// Mitsubishi GX Works2 project: PLC_GROUP9   PLC: FX3G

// global labels: Global1
VAR_GLOBAL
  init AT X010 : BOOL;
END_VAR
VAR_GLOBAL CONSTANT
  OrangeValue : REAL;
END_VAR
VAR_GLOBAL
  RE_initOrange AT D1100 : REAL;
END_VAR
VAR_GLOBAL CONSTANT
  ClementineValue : REAL;
END_VAR
VAR_GLOBAL
  RE_initClem AT D1120 : REAL;
END_VAR
VAR_GLOBAL CONSTANT
  PomeloValue : REAL;
END_VAR
VAR_GLOBAL
  RE_initPomeo AT D1110 : REAL;
  Sw10 AT X010 : BOOL;
END_VAR
VAR_GLOBAL CONSTANT
  CorrectDiv : INT := 2;
END_VAR
VAR_GLOBAL
  RE_CorrectDiv AT D1115 : REAL;
END_VAR
VAR_GLOBAL CONSTANT
  HelpValue : INT := 1;
END_VAR
VAR_GLOBAL
  StopWork AT X007 : BOOL;
END_VAR
VAR_GLOBAL CONSTANT
  two : REAL := 2.0;
END_VAR
VAR_GLOBAL
  ClementineOn AT M0 : BOOL;
  PomeloOn AT M1 : BOOL;
  bulb1 AT Y010 : BOOL;
END_VAR
VAR_GLOBAL CONSTANT
  zero : REAL;
END_VAR
VAR_GLOBAL
  RE_Orange AT D1150 : REAL;
  RE_Clem AT D1130 : REAL;
  RE_Pomelo AT D1140 : REAL;
  SystemOn AT M2 : BOOL;
  bnnb AT M3 : BOOL;
  m_6 AT M7 : BOOL;
  StartingValuesOn AT M0 : BOOL;
  InventoryValuesOn AT M1 : BOOL;
  SystemOff AT M2 : BOOL;
  SystemOf AT M2 : BOOL;
  StopConditions AT M3 : BOOL;
  FlashingLight1 AT M4 : BOOL;
  FlickeringTimer1 AT TC0 : BOOL;
END_VAR
VAR_GLOBAL CONSTANT
  VNBVNBV : INT := 30;
  ConstantFlickering1 : INT := 5;
END_VAR
VAR_GLOBAL
  TimerValue1 AT TS0 : BOOL;
  FlickeringLight1 AT M4 : BOOL;
  FlickeringLight2 AT M5 : BOOL;
  FlickeringTimer2 AT TC1 : BOOL;
  TimerValue2 AT TS1 : BOOL;
  FlickeringLightStop AT M6 : BOOL;
  FlickeringTimer3 AT TC2 : BOOL;
  FlickeringStoper AT TS2 : BOOL;
END_VAR
VAR_GLOBAL CONSTANT
  Var_Time_0 : INT := 30;
END_VAR
VAR_GLOBAL
  Constant_300 AT K3 : INT;
  Washing_help AT M10 : BOOL;
  Start AT M10 : BOOL;
  Start_Washing AT X002 : BOOL;
  light_on AT M11 : BOOL;
  Close_light AT TS3 : BOOL;
  Start_light AT M10 : BOOL;
  bulb5 AT Y005 : BOOL;
  Start_Wash AT M10 : BOOL;
END_VAR
VAR_GLOBAL CONSTANT
  Constant_100 : REAL := 100;
END_VAR
VAR_GLOBAL
  More_100 AT M12 : BOOL;
  Washing_Orange AT D1170 : REAL;
  over_100_ans AT M13 : BOOL;
END_VAR
VAR_GLOBAL CONSTANT
  Constant_2 : REAL := 2;
END_VAR
VAR_GLOBAL
  Quantity_To_Move AT D1180 : REAL;
  Finish_Orange AT M15 : BOOL;
  Washing_Clem AT D1190 : REAL;
  Washing_Pomalo AT D1200 : REAL;
  under_100_ans AT M14 : BOOL;
  orange_ans AT M13 : BOOL;
END_VAR
VAR_GLOBAL CONSTANT
  ConstantFlickering : INT := 30;
END_VAR
VAR_GLOBAL
  StartCounter AT CC0 : BOOL;
END_VAR
VAR_GLOBAL CONSTANT
  CounterStert : INT := 3;
  CounterStart : INT := 1;
END_VAR
VAR_GLOBAL
  StertDay AT CS0 : BOOL;
  not1 AT M30 : BOOL;
  not2 AT M31 : BOOL;
  Timer3 AT TC3 : BOOL;
END_VAR
VAR_GLOBAL CONSTANT
  ConstantWashing : INT := 30;
END_VAR
VAR_GLOBAL
  End_level1 AT M16 : BOOL;
END_VAR
VAR_GLOBAL CONSTANT
  DubbleClick : INT := 2;
END_VAR
VAR_GLOBAL
  Start_level_Two AT CC1 : BOOL;
  Start_Collect AT X001 : BOOL;
  Start_Collect_SW AT X011 : BOOL;
  Collect_light AT Y001 : BOOL;
  Squeeze_SW AT X011 : BOOL;
  Squeezing : BOOL;
  Start_squeezing AT CS1 : BOOL;
  Start_level_Three AT CC1 : BOOL;
  SqueezeContainer AT D2200 : REAL;
  Finish_move AT M17 : BOOL;
  End_level2 AT M18 : BOOL;
  helpBulb AT M19 : BOOL;
  helpBulb2 AT M20 : BOOL;
  level_Three AT CS1 : BOOL;
  kkkk AT Y002 : BOOL;
  Timer4 AT TC4 : BOOL;
  Stop_Flickering AT TS4 : BOOL;
  SqueezeLight1 AT Y002 : BOOL;
  SqueezeLight2 AT Y003 : BOOL;
  JoiceContainer AT D1210 : REAL;
  JuiceContainer AT D1210 : REAL;
  End_level3 AT M32 : BOOL;
  helpBulb3 AT M41 : BOOL;
  Start_level_four AT X003 : BOOL;
  helpBulb4 AT M34 : BOOL;
  Start_Quality_Check AT X003 : BOOL;
  Failed_Check AT M38 : BOOL;
  Start_level_4 AT M35 : BOOL;
  Finish_level_three AT M40 : BOOL;
  Secend_Check AT CS5 : BOOL;
  Counter_Check AT CC5 : BOOL;
END_VAR
VAR_GLOBAL CONSTANT
  Limit_Check : INT := 2;
END_VAR
VAR_GLOBAL
  analog_input_2 AT D8281 : INT;
  analog_val AT D1300 : INT;
END_VAR
VAR_GLOBAL CONSTANT
  Constant_1 : INT := 1;
END_VAR
VAR_GLOBAL
  helpBulb6 AT M37 : BOOL;
END_VAR
VAR_GLOBAL CONSTANT
  Constant_5 : INT := 4;
END_VAR
VAR_GLOBAL
  helpBulbEnd3 AT M33 : BOOL;
  need_restart AT M39 : BOOL;
  FlickeringStoper5 AT TS5 : BOOL;
  Val_In_Range AT Y004 : BOOL;
  FlickeringTimer5 AT TC5 : BOOL;
END_VAR
VAR_GLOBAL CONSTANT
  ConstantFlickering5 : INT := 50;
END_VAR
VAR_GLOBAL
  Start_Container AT M41 : BOOL;
  Storage_Container AT D1320 : REAL;
  End_level4 AT M42 : BOOL;
  End_day AT M31 : BOOL;
  MoreThen1 AT M44 : BOOL;
  LessThen5 AT M45 : BOOL;
  ValBulb AT M46 : BOOL;
  Stoper AT CS0 : BOOL;
  endBulb1 AT M47 : BOOL;
  endBulb2 AT M48 : BOOL;
  endBulb3 AT M49 : BOOL;
  endBulb4 AT M50 : BOOL;
  Endbulb5 AT M51 : BOOL;
END_VAR
VAR_GLOBAL CONSTANT
  Constant_3c : REAL := 20;
END_VAR
VAR_GLOBAL
  Enough_Liter AT M57 : BOOL;
END_VAR
VAR_GLOBAL CONSTANT
  Constant_3 : REAL := 20;
END_VAR
VAR_GLOBAL
  Analog_Output AT D8282 : INT;
  Finish_Count AT M62 : BOOL;
  FlickeringTimer6 AT TC6 : BOOL;
  FlickeringStoper6 AT TS6 : BOOL;
  StartToBottle AT X006 : BOOL;
  End_level5 AT M60 : BOOL;
  notEnoughJuice AT M61 : BOOL;
  Timer6 AT TC6 : BOOL;
  StoperTimer6 AT TS6 : BOOL;
  NotBottle AT Y006 : BOOL;
END_VAR
VAR_GLOBAL CONSTANT
  ConvertingCon : INT := 404;
  Constant_10c : REAL := 20;
  Constant_20c : REAL := 20;
END_VAR
VAR_GLOBAL
  bulb1ForRest AT M70 : BOOL;
  bulb2ForRest AT M71 : BOOL;
  CheckStartCon AT M72 : BOOL;
  QuantityPerIteration AT D1340 : REAL;
  StartContainer AT CC0 : BOOL;
  StartToContainer AT X006 : BOOL;
  NotContainer AT Y006 : BOOL;
END_VAR
VAR_GLOBAL CONSTANT
  notEnough : INT;
END_VAR

// task Task_01 (event TRUE, interval 0, priority 31): POU_01

PROGRAM POU_01
(* structured ladder/FBD written out as ST: instructions are called as NAME(EN, inputs, outputs); _pN, _eN, _tN stand for wires *)
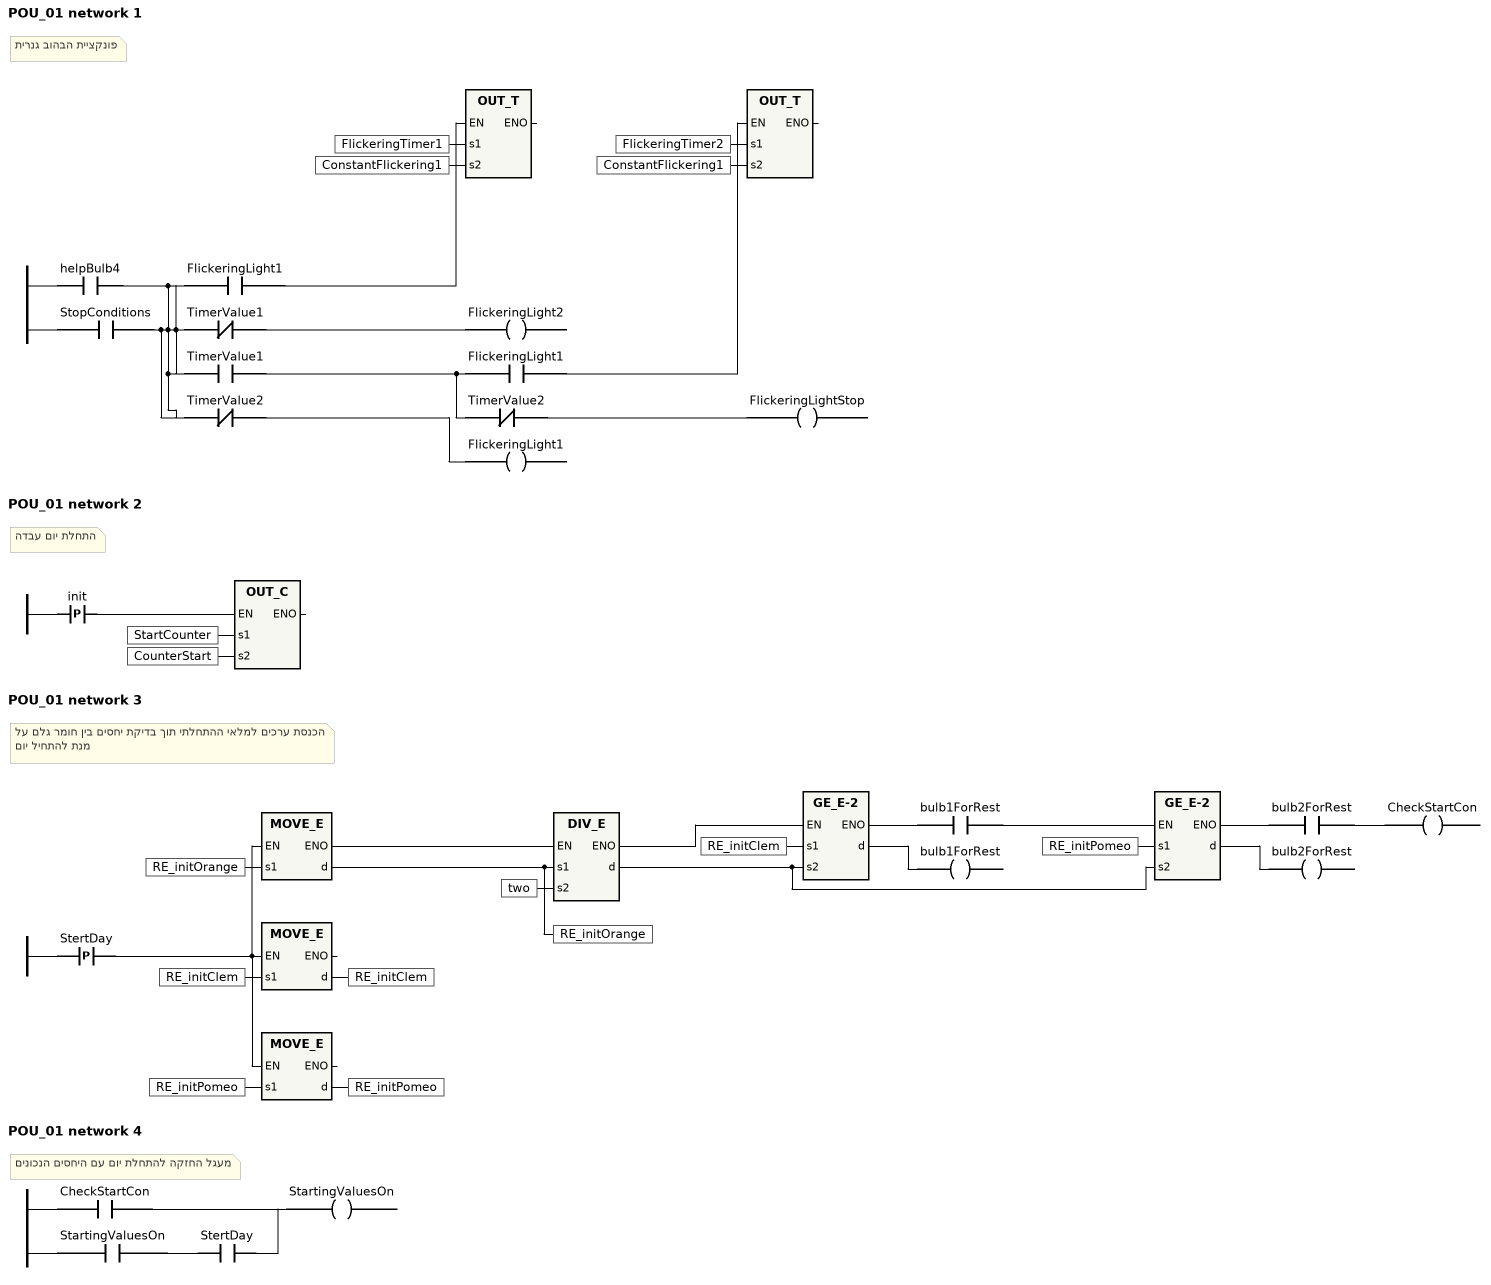
(* network 1 *)
(* פונקציית הבהוב גנרית *)
_p1 := helpBulb4 OR StopConditions;
OUT_T(_p1 AND FlickeringLight1, FlickeringTimer1, ConstantFlickering1);
FlickeringLight2 := _p1 AND NOT TimerValue1;
_p2 := _p1 AND TimerValue1;
OUT_T(_p2 AND FlickeringLight1, FlickeringTimer2, ConstantFlickering1);
FlickeringLightStop := _p2 AND NOT TimerValue2;
FlickeringLight1 := _p1 AND NOT TimerValue2;
(* network 2 *)
(* התחלת יום עבדה *)
OUT_C(LDP(TRUE, init), StartCounter, CounterStart);
(* network 3 *)
(* הכנסת ערכים למלאי ההתחלתי תוך בדיקת יחסים בין חומר גלם על מנת להתחיל יום *)
_p1 := LDP(TRUE, StertDay);
_e2 := MOVE_E(_p1, RE_initOrange, RE_initOrange);
_e4 := DIV_E(_e2, RE_initOrange, two, _t3);
_e6 := GE_E(_e4, RE_initClem, _t3, _t5);
bulb1ForRest := _t5;
MOVE_E(_p1, RE_initClem, RE_initClem);
_e8 := GE_E(_e6 AND bulb1ForRest, RE_initPomeo, _t3, _t7);
CheckStartCon := _e8 AND bulb2ForRest;
MOVE_E(_p1, RE_initPomeo, RE_initPomeo);
bulb2ForRest := _t7;
(* network 4 *)
(* מעגל החזקה להתחלת יום עם היחסים הנכונים *)
StartingValuesOn := CheckStartCon OR (StartingValuesOn AND StertDay);
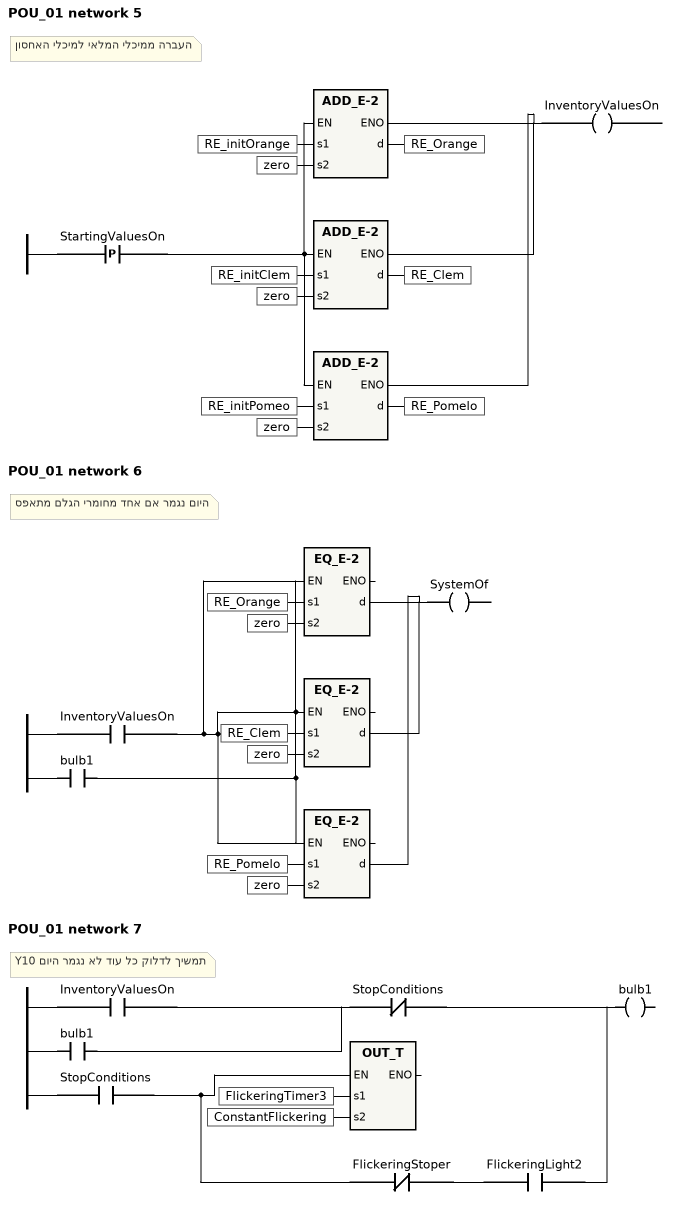
(* network 5 *)
(* העברה ממיכלי המלאי למיכלי האחסון *)
_p1 := LDP(TRUE, StartingValuesOn);
_e2 := ADD_E(_p1, RE_initOrange, zero, RE_Orange);
_e3 := ADD_E(_p1, RE_initClem, zero, RE_Clem);
_e4 := ADD_E(_p1, RE_initPomeo, zero, RE_Pomelo);
InventoryValuesOn := _e2 OR _e3 OR _e4;
(* network 6 *)
(* היום נגמר אם אחד מחומרי הגלם מתאפס *)
_p1 := InventoryValuesOn OR bulb1;
EQ_E(_p1, RE_Orange, zero, _t2);
EQ_E(_p1, RE_Clem, zero, _t3);
EQ_E(_p1, RE_Pomelo, zero, _t4);
SystemOf := _t2 OR _t3 OR _t4;
(* network 7 *)
(* תמשיך לדלוק כל עוד לא נגמר היום Y10 *)
bulb1 := ((InventoryValuesOn OR bulb1) AND NOT StopConditions) OR (StopConditions AND NOT FlickeringStoper AND FlickeringLight2);
OUT_T(StopConditions, FlickeringTimer3, ConstantFlickering);
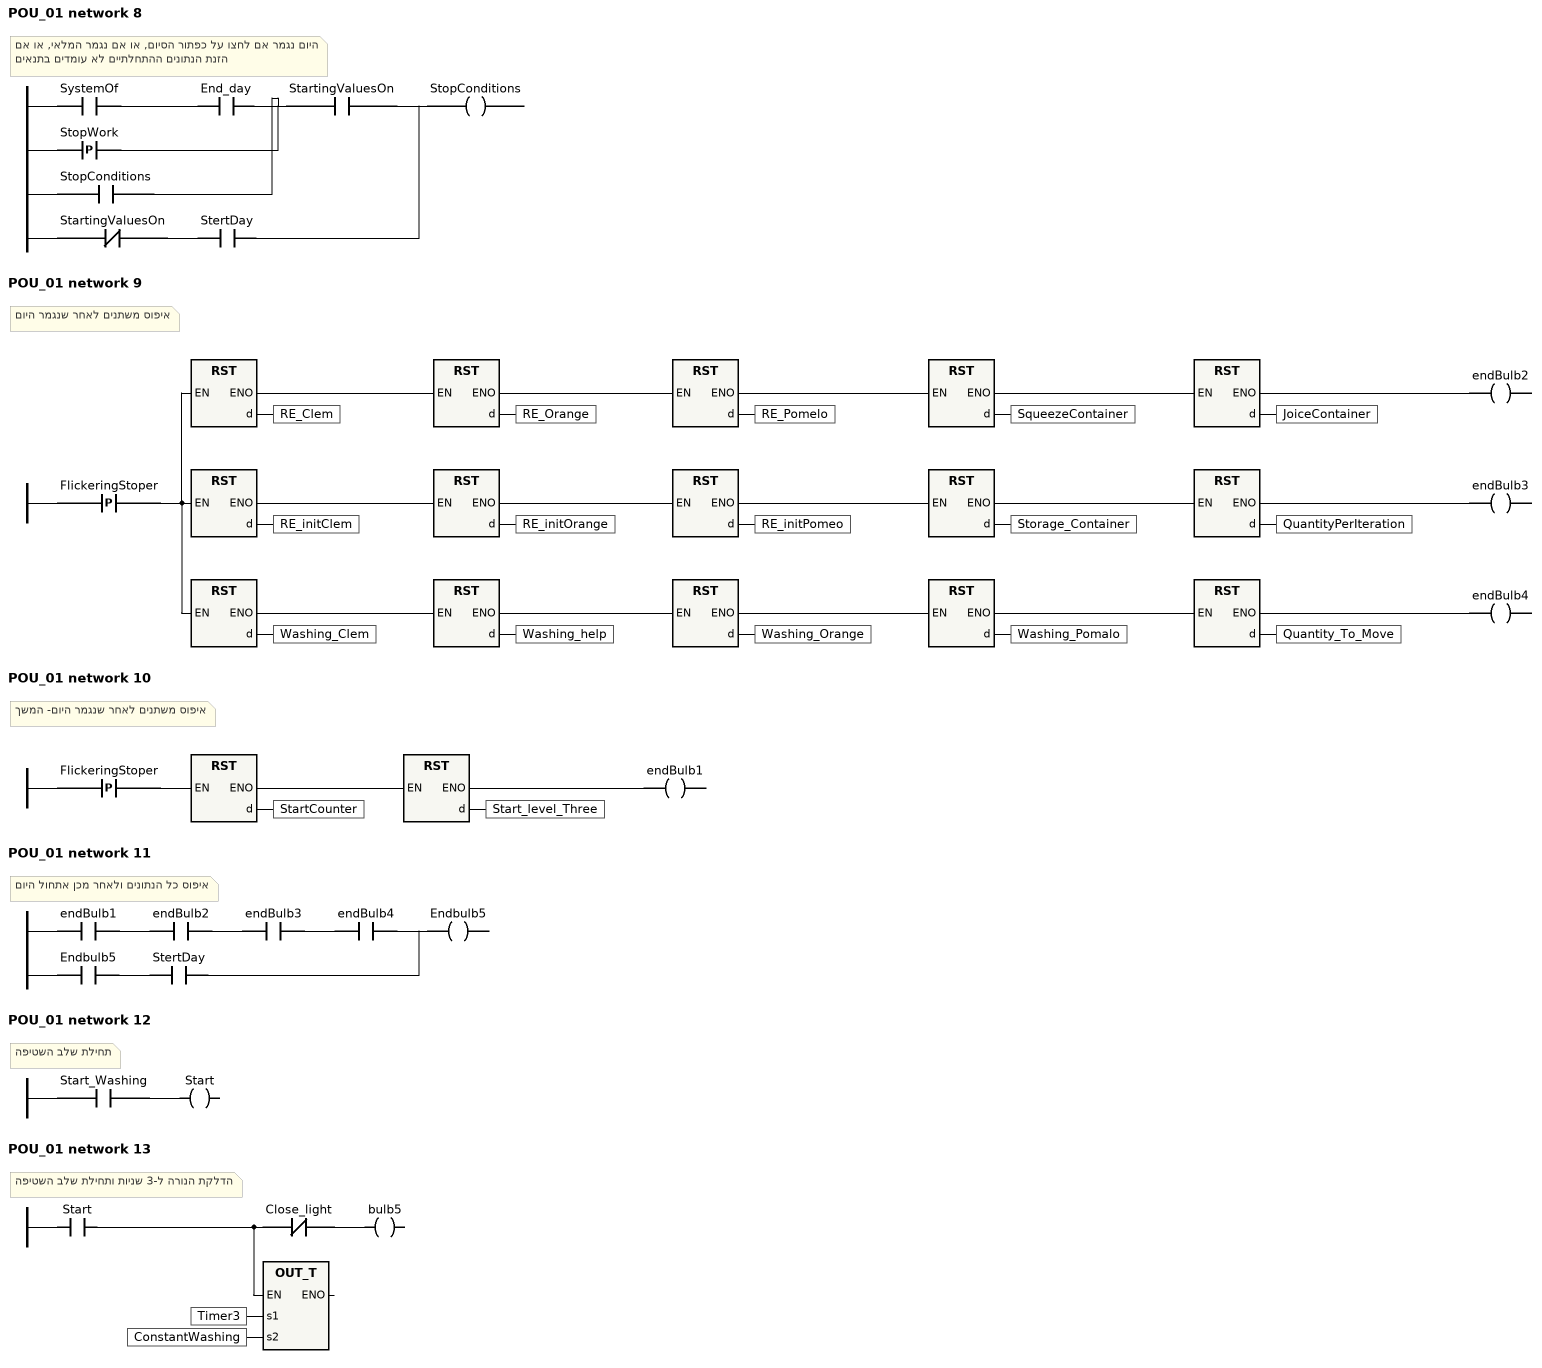
(* network 8 *)
(* היום נגמר אם לחצו על כפתור הסיום, או אם נגמר המלאי, או אם הזנת הנתונים ההתחלתיים לא עומדים בתנאים *)
StopConditions := (((SystemOf AND End_day) OR LDP(TRUE, StopWork) OR StopConditions) AND StartingValuesOn) OR (NOT StartingValuesOn AND StertDay);
(* network 9 *)
(* איפוס משתנים לאחר שנגמר היום *)
_p1 := LDP(TRUE, FlickeringStoper);
_e2 := RST(_p1, RE_Clem);
_e3 := RST(_e2, RE_Orange);
_e4 := RST(_e3, RE_Pomelo);
_e5 := RST(_e4, SqueezeContainer);
_e6 := RST(_e5, JoiceContainer);
endBulb2 := _e6;
_e7 := RST(_p1, RE_initClem);
_e8 := RST(_e7, RE_initOrange);
_e9 := RST(_e8, RE_initPomeo);
_e10 := RST(_e9, Storage_Container);
_e11 := RST(_e10, QuantityPerIteration);
endBulb3 := _e11;
_e12 := RST(_p1, Washing_Clem);
_e13 := RST(_e12, Washing_help);
_e14 := RST(_e13, Washing_Orange);
_e15 := RST(_e14, Washing_Pomalo);
_e16 := RST(_e15, Quantity_To_Move);
endBulb4 := _e16;
(* network 10 *)
(* איפוס משתנים לאחר שנגמר היום- המשך *)
_e1 := RST(LDP(TRUE, FlickeringStoper), StartCounter);
_e2 := RST(_e1, Start_level_Three);
endBulb1 := _e2;
(* network 11 *)
(* איפוס כל הנתונים ולאחר מכן אתחול היום *)
Endbulb5 := (endBulb1 AND endBulb2 AND endBulb3 AND endBulb4) OR (Endbulb5 AND StertDay);
(* network 12 *)
(* תחילת שלב השטיפה *)
Start := Start_Washing;
(* network 13 *)
(* הדלקת הנורה ל-3 שניות ותחילת שלב השטיפה *)
bulb5 := Start AND NOT Close_light;
OUT_T(Start, Timer3, ConstantWashing);
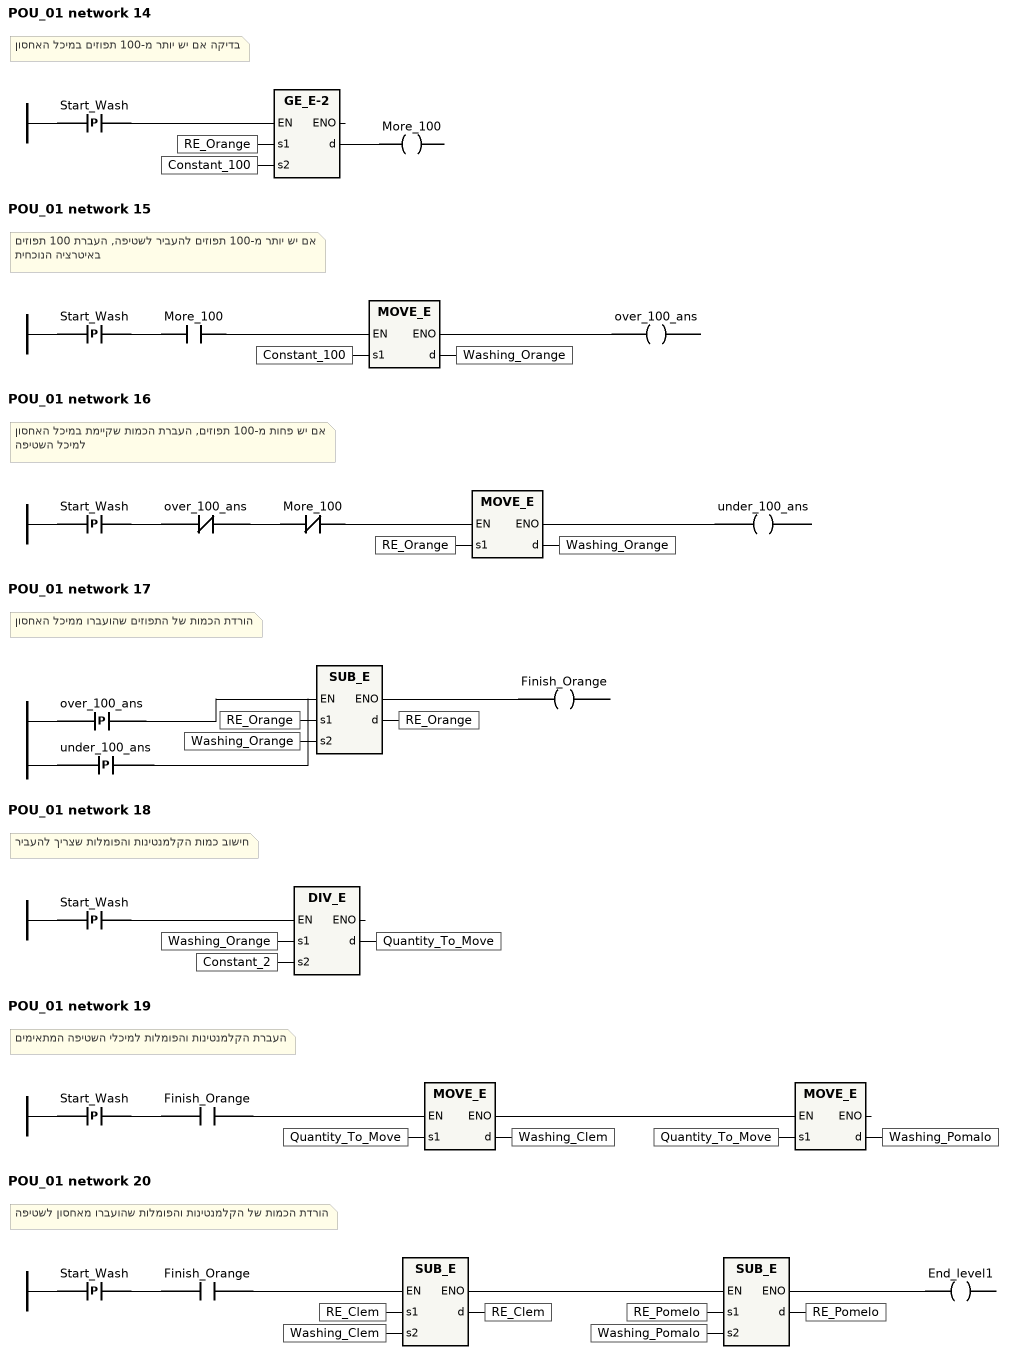
(* network 14 *)
(* בדיקה אם יש יותר מ-100 תפוזים במיכל האחסון *)
GE_E(LDP(TRUE, Start_Wash), RE_Orange, Constant_100, _t1);
More_100 := _t1;
(* network 15 *)
(* אם יש יותר מ-100 תפוזים להעביר לשטיפה, העברת 100 תפוזים באיטרציה הנוכחית *)
_e1 := MOVE_E(LDP(TRUE, Start_Wash) AND More_100, Constant_100, Washing_Orange);
over_100_ans := _e1;
(* network 16 *)
(* אם יש פחות מ-100 תפוזים, העברת הכמות שקיימת במיכל האחסון למיכל השטיפה *)
_e1 := MOVE_E(LDP(TRUE, Start_Wash) AND NOT over_100_ans AND NOT More_100, RE_Orange, Washing_Orange);
under_100_ans := _e1;
(* network 17 *)
(* הורדת הכמות של התפוזים שהועברו ממיכל האחסון *)
_e1 := SUB_E(LDP(TRUE, over_100_ans) OR LDP(TRUE, under_100_ans), RE_Orange, Washing_Orange, RE_Orange);
Finish_Orange := _e1;
(* network 18 *)
(* חישוב כמות הקלמנטינות והפומלות שצריך להעביר *)
DIV_E(LDP(TRUE, Start_Wash), Washing_Orange, Constant_2, Quantity_To_Move);
(* network 19 *)
(* העברת הקלמנטינות והפומלות למיכלי השטיפה המתאימים *)
_e1 := MOVE_E(LDP(TRUE, Start_Wash) AND Finish_Orange, Quantity_To_Move, Washing_Clem);
MOVE_E(_e1, Quantity_To_Move, Washing_Pomalo);
(* network 20 *)
(* הורדת הכמות של הקלמנטינות והפומלות שהועברו מאחסון לשטיפה *)
_e1 := SUB_E(LDP(TRUE, Start_Wash) AND Finish_Orange, RE_Clem, Washing_Clem, RE_Clem);
_e2 := SUB_E(_e1, RE_Pomelo, Washing_Pomalo, RE_Pomelo);
End_level1 := _e2;
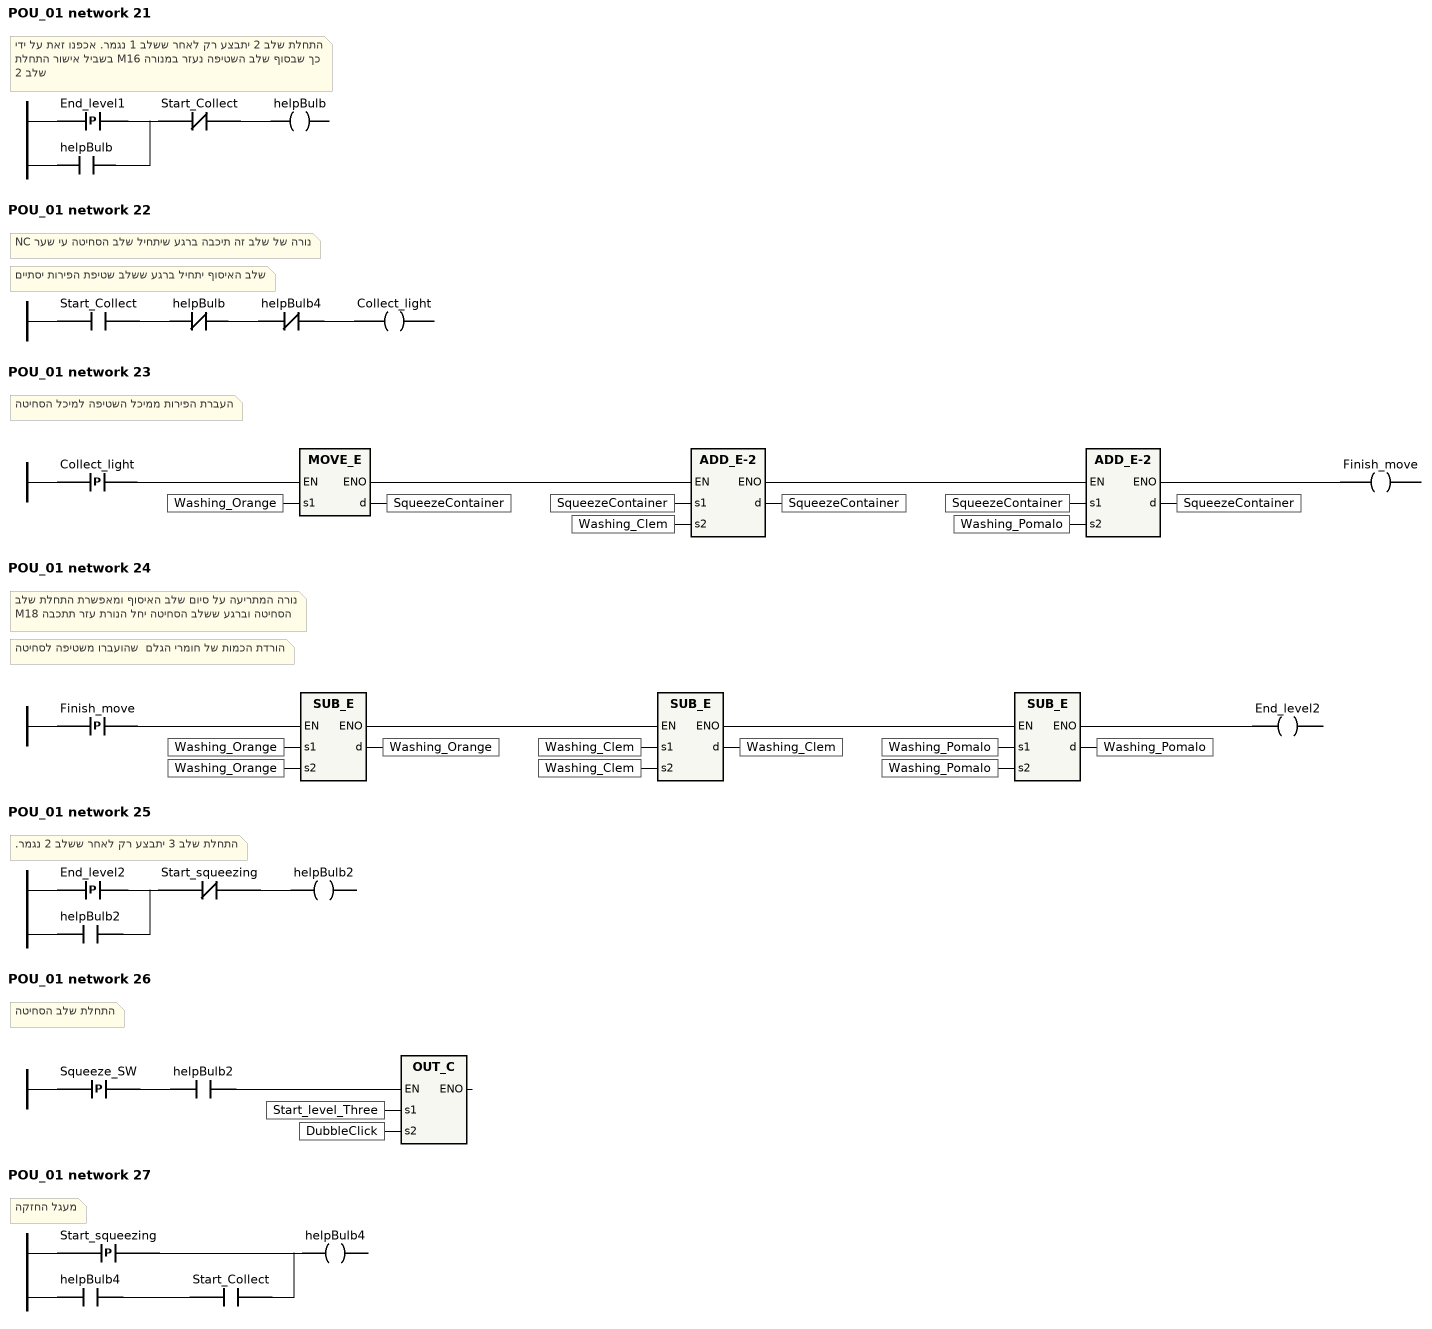
(* network 21 *)
(* התחלת שלב 2 יתבצע רק לאחר ששלב 1 נגמר. אכפנו זאת על ידי  כך שבסוף שלב השטיפה נעזר במנורה M16 בשביל אישור התחלת שלב 2 *)
helpBulb := (LDP(TRUE, End_level1) OR helpBulb) AND NOT Start_Collect;
(* network 22 *)
(* נורה של שלב זה תיכבה ברגע שיתחיל שלב הסחיטה עי שער NC *)
(* שלב האיסוף יתחיל ברגע ששלב שטיפת הפירות יסתיים *)
Collect_light := Start_Collect AND NOT helpBulb AND NOT helpBulb4;
(* network 23 *)
(* העברת הפירות ממיכל השטיפה למיכל הסחיטה *)
_e1 := MOVE_E(LDP(TRUE, Collect_light), Washing_Orange, SqueezeContainer);
_e2 := ADD_E(_e1, SqueezeContainer, Washing_Clem, SqueezeContainer);
_e3 := ADD_E(_e2, SqueezeContainer, Washing_Pomalo, SqueezeContainer);
Finish_move := _e3;
(* network 24 *)
(* נורה המתריעה על סיום שלב האיסוף ומאפשרת התחלת שלב הסחיטה וברגע ששלב הסחיטה יחל הנורת עזר תתכבה M18 *)
(* הורדת הכמות של חומרי הגלם  שהועברו משטיפה לסחיטה *)
_e1 := SUB_E(LDP(TRUE, Finish_move), Washing_Orange, Washing_Orange, Washing_Orange);
_e2 := SUB_E(_e1, Washing_Clem, Washing_Clem, Washing_Clem);
_e3 := SUB_E(_e2, Washing_Pomalo, Washing_Pomalo, Washing_Pomalo);
End_level2 := _e3;
(* network 25 *)
(* התחלת שלב 3 יתבצע רק לאחר ששלב 2 נגמר. *)
helpBulb2 := (LDP(TRUE, End_level2) OR helpBulb2) AND NOT Start_squeezing;
(* network 26 *)
(* התחלת שלב הסחיטה *)
OUT_C(LDP(TRUE, Squeeze_SW) AND helpBulb2, Start_level_Three, DubbleClick);
(* network 27 *)
(* מעגל החזקה *)
helpBulb4 := LDP(TRUE, Start_squeezing) OR (helpBulb4 AND Start_Collect);
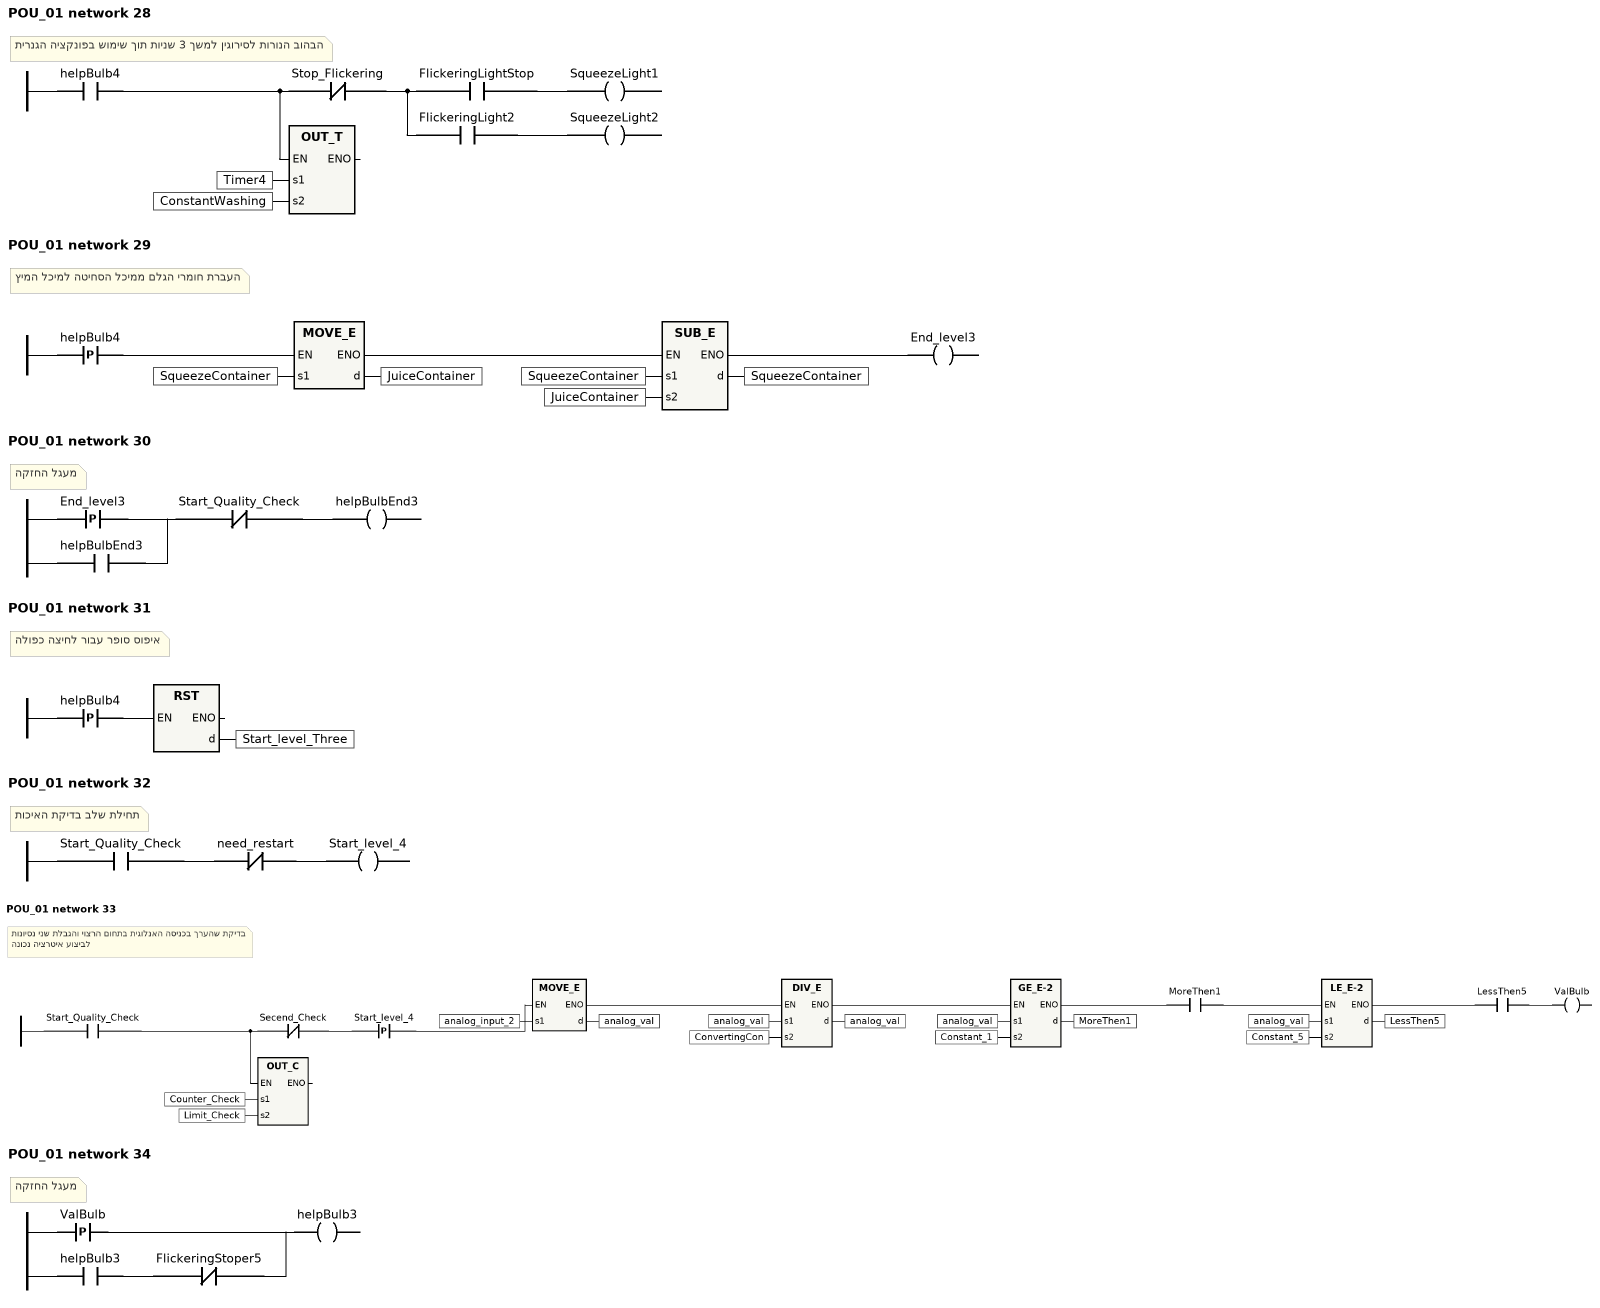
(* network 28 *)
(* הבהוב הנורות לסירוגין למשך 3 שניות תוך שימוש בפונקציה הגנרית *)
_p1 := helpBulb4 AND NOT Stop_Flickering;
SqueezeLight1 := _p1 AND FlickeringLightStop;
SqueezeLight2 := _p1 AND FlickeringLight2;
OUT_T(helpBulb4, Timer4, ConstantWashing);
(* network 29 *)
(* העברת חומרי הגלם ממיכל הסחיטה למיכל המיץ *)
_e1 := MOVE_E(LDP(TRUE, helpBulb4), SqueezeContainer, JuiceContainer);
_e2 := SUB_E(_e1, SqueezeContainer, JuiceContainer, SqueezeContainer);
End_level3 := _e2;
(* network 30 *)
(* מעגל החזקה *)
helpBulbEnd3 := (LDP(TRUE, End_level3) OR helpBulbEnd3) AND NOT Start_Quality_Check;
(* network 31 *)
(* איפוס סופר עבור לחיצה כפולה *)
RST(LDP(TRUE, helpBulb4), Start_level_Three);
(* network 32 *)
(* תחילת שלב בדיקת האיכות *)
Start_level_4 := Start_Quality_Check AND NOT need_restart;
(* network 33 *)
(* בדיקת שהערך בכניסה האנלוגית בתחום הרצוי והגבלת שני נסיונות לביצוע איטרציה נכונה *)
_e1 := MOVE_E(Start_Quality_Check AND NOT Secend_Check AND LDP(TRUE, Start_level_4), analog_input_2, analog_val);
_e2 := DIV_E(_e1, analog_val, ConvertingCon, analog_val);
_e3 := GE_E(_e2, analog_val, Constant_1, MoreThen1);
_e4 := LE_E(_e3 AND MoreThen1, analog_val, Constant_5, LessThen5);
ValBulb := _e4 AND LessThen5;
OUT_C(Start_Quality_Check, Counter_Check, Limit_Check);
(* network 34 *)
(* מעגל החזקה *)
helpBulb3 := LDP(TRUE, ValBulb) OR (helpBulb3 AND NOT FlickeringStoper5);
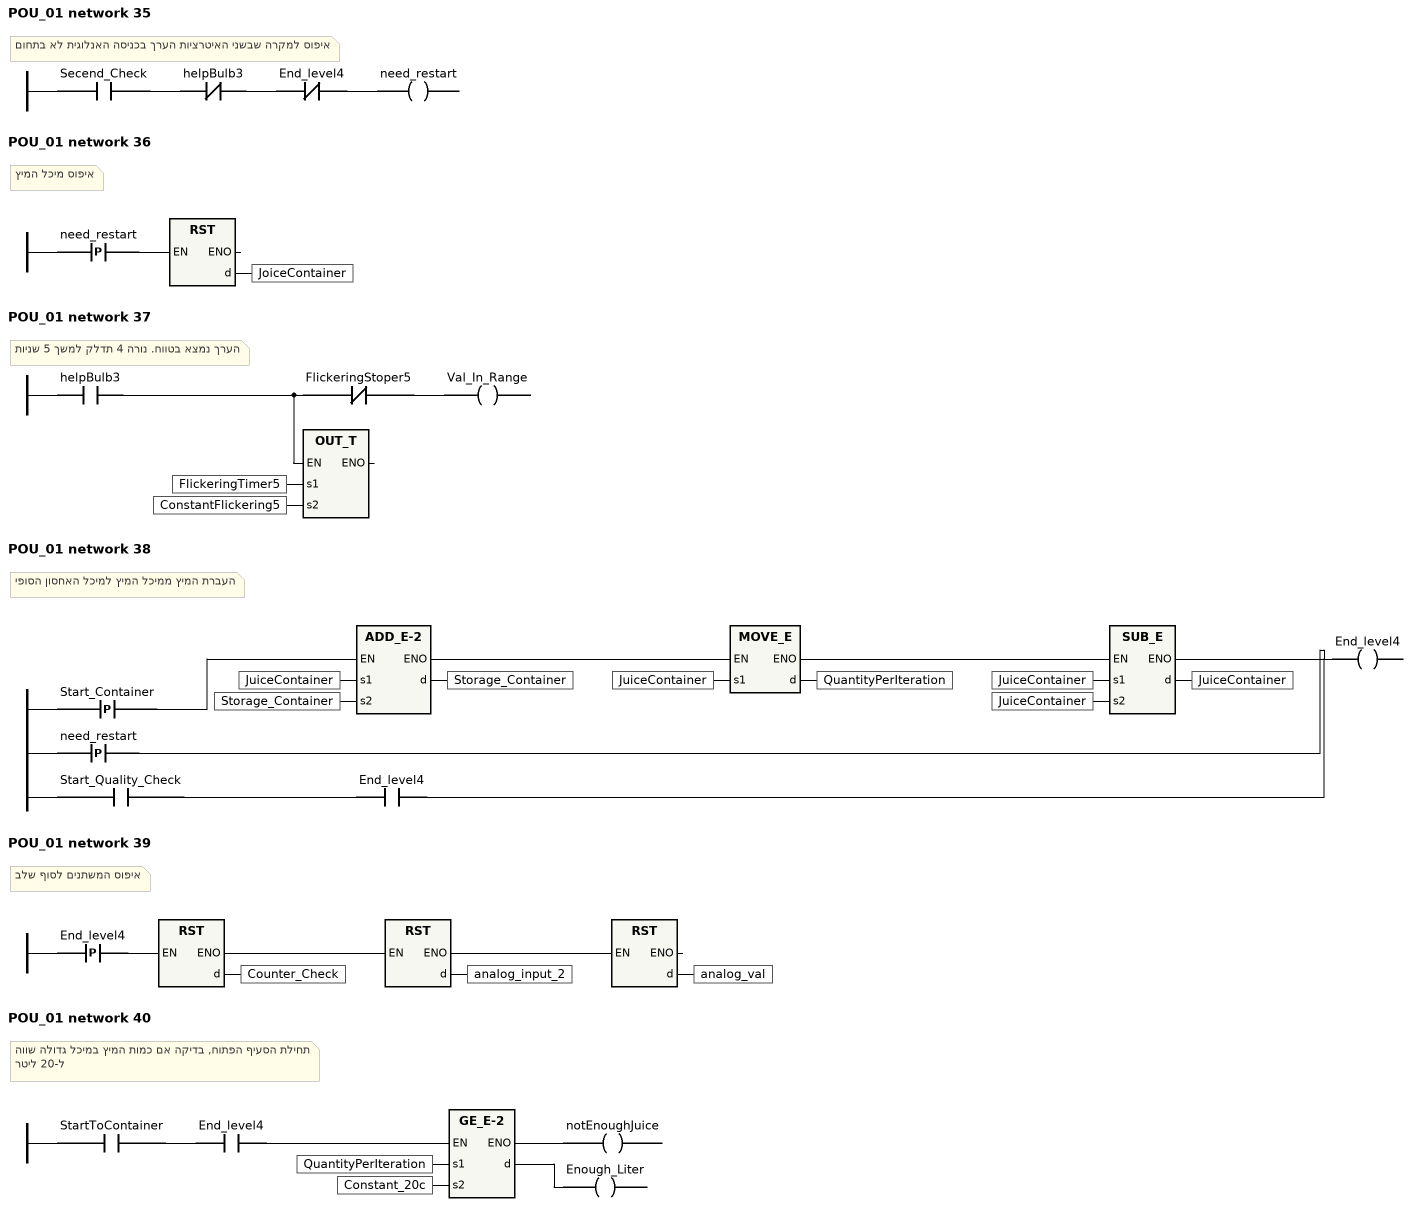
(* network 35 *)
(* איפוס למקרה שבשני האיטרציות הערך בכניסה האנלוגית לא בתחום *)
need_restart := Secend_Check AND NOT helpBulb3 AND NOT End_level4;
(* network 36 *)
(* איפוס מיכל המיץ *)
RST(LDP(TRUE, need_restart), JoiceContainer);
(* network 37 *)
(* הערך נמצא בטווח. נורה 4 תדלק למשך 5 שניות *)
Val_In_Range := helpBulb3 AND NOT FlickeringStoper5;
OUT_T(helpBulb3, FlickeringTimer5, ConstantFlickering5);
(* network 38 *)
(* העברת המיץ ממיכל המיץ למיכל האחסון הסופי *)
_e1 := ADD_E(LDP(TRUE, Start_Container), JuiceContainer, Storage_Container, Storage_Container);
_e2 := MOVE_E(_e1, JuiceContainer, QuantityPerIteration);
_e3 := SUB_E(_e2, JuiceContainer, JuiceContainer, JuiceContainer);
End_level4 := _e3 OR LDP(TRUE, need_restart) OR (Start_Quality_Check AND End_level4);
(* network 39 *)
(* איפוס המשתנים לסוף שלב *)
_e1 := RST(LDP(TRUE, End_level4), Counter_Check);
_e2 := RST(_e1, analog_input_2);
RST(_e2, analog_val);
(* network 40 *)
(* תחילת הסעיף הפתוח, בדיקה אם כמות המיץ במיכל גדולה שווה ל-20 ליטר *)
_e2 := GE_E(StartToContainer AND End_level4, QuantityPerIteration, Constant_20c, _t1);
notEnoughJuice := _e2;
Enough_Liter := _t1;
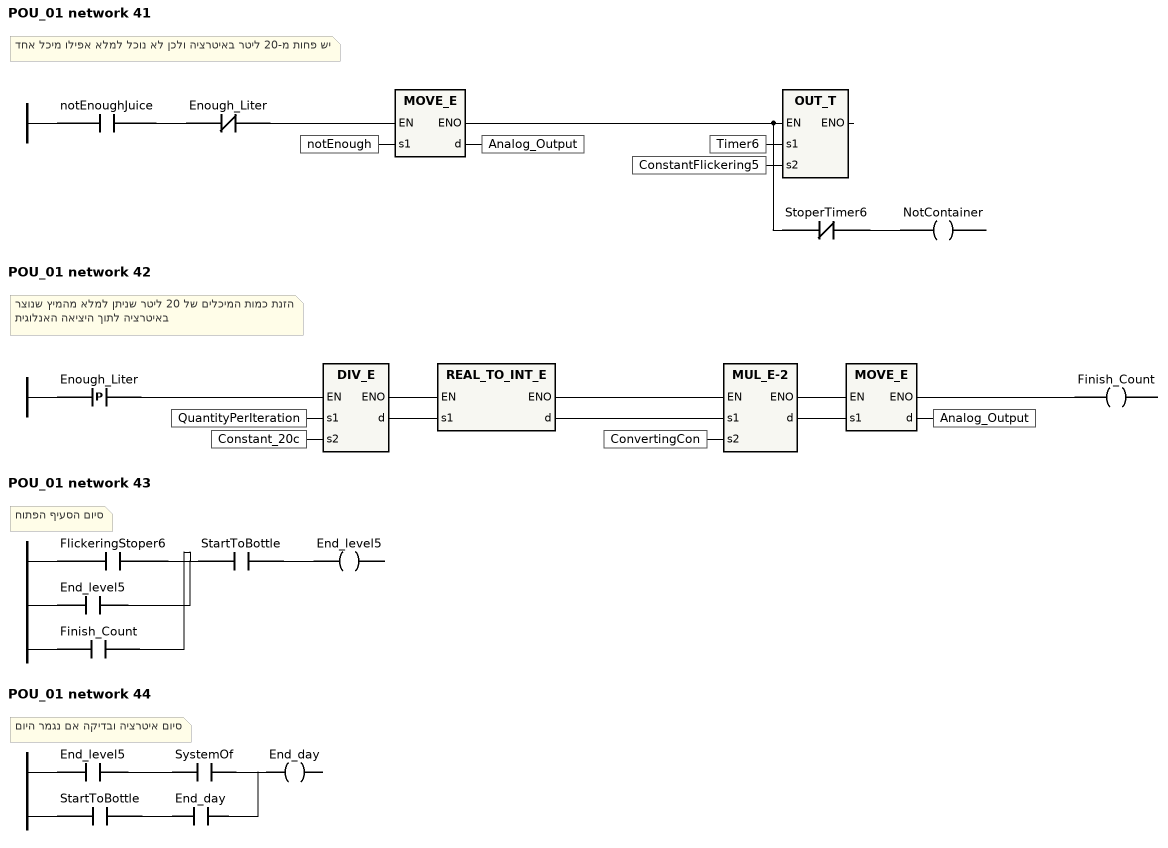
(* network 41 *)
(* יש פחות מ-20 ליטר באיטרציה ולכן לא נוכל למלא אפילו מיכל אחד *)
_e1 := MOVE_E(notEnoughJuice AND NOT Enough_Liter, notEnough, Analog_Output);
NotContainer := _e1 AND NOT StoperTimer6;
OUT_T(_e1, Timer6, ConstantFlickering5);
(* network 42 *)
(* הזנת כמות המיכלים של 20 ליטר שניתן למלא מהמיץ שנוצר באיטרציה לתוך היציאה האנלוגית *)
_e2 := DIV_E(LDP(TRUE, Enough_Liter), QuantityPerIteration, Constant_20c, _t1);
_e4 := REAL_TO_INT_E(_e2, _t1, _t3);
_e6 := MUL_E(_e4, _t3, ConvertingCon, _t5);
_e7 := MOVE_E(_e6, _t5, Analog_Output);
Finish_Count := _e7;
(* network 43 *)
(* סיום הסעיף הפתוח *)
End_level5 := (FlickeringStoper6 OR End_level5 OR Finish_Count) AND StartToBottle;
(* network 44 *)
(* סיום איטרציה ובדיקה אם נגמר היום *)
End_day := (End_level5 AND SystemOf) OR (StartToBottle AND End_day);
END_PROGRAM
